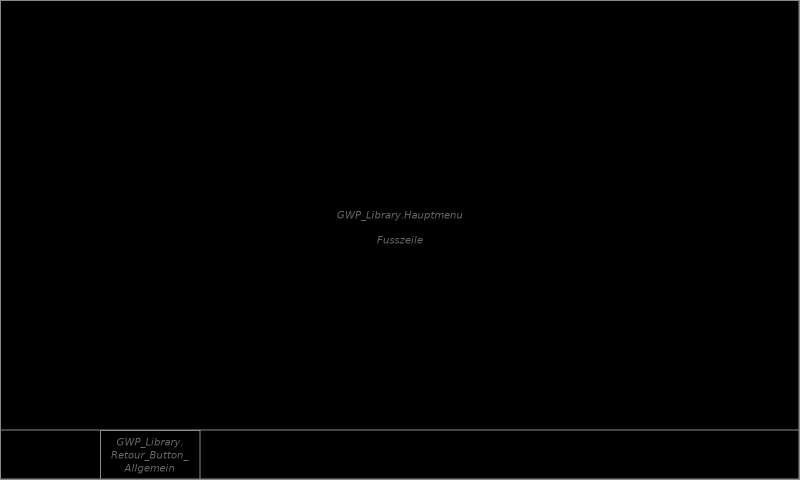
VISUALIZATION Menue  // 800x480
    Frame (0,0 800x480)
        shows Fusszeile()
    Frame (100,430 100x50)
        shows GWP_Library.Retour_Button_Allgemein()
    Frame (0,0 800x430)
        shows GWP_Library.Hauptmenu(FB_Init_1 := MAIN.Init_0)
END_VISUALIZATION

(* stored: Version 1.1.0.1, ProductVersion 3.1.4022.6
   Visu Menue: Id {4b340ce0-0596-4a34-a052-60c0db83a469} *)
